# EPICS autosave request: dxpApp/Db/microDXP_settings.req
$(P)$(R)Gain
$(P)$(R)FineGain
